// TIA Portal V16 export
// export: Created 2020-08-26T14:42:00.343357Z, ExportSetting WithDefaults, DisplayName Totally Integrated Automation Portal, DisplayVersion V16 Update 2, DisplayName TIA Portal Version Control Interface, DisplayVersion V16 Update 2, DisplayName TIA Portal Openness, DisplayVersion V16 Update 2, DisplayName TIA Portal Teamcenter Gateway, DisplayVersion V16, DisplayName SINAMICS Startdrive Advanced, DisplayVersion V16 Update 1, DisplayName SINAMICS Startdrive G130, G150, S120, S150, SINAMICS MV, S210, DisplayVersion V16 Update 1, DisplayName SINAMICS Startdrive G110M, G120, G120C, G120D, G120P, DisplayVersion V16 Update 1, DisplayName STEP 7 Professional, DisplayVersion V16 Update 2, DisplayName SIMATIC Energy Suite, DisplayVersion V16, DisplayName STEP 7 Safety, DisplayVersion V16, DisplayName WinCC Professional, DisplayVersion V16 Update 2
FUNCTION_BLOCK "SimpleMotor"   // FB2, LAD
{ S7_Optimized_Access := 'TRUE' }
VERSION : 0.1
// stored: AutoNumber true, IsIECCheckEnabled false, IsRetainMemResEnabled false, MemoryReserve 100, SetENOAutomatically false, UDAEnableTagReadback false
   VAR_INPUT
      Start : Bool;
      Stop : Bool;
      Overload : Bool;
      Fault : Bool;
      Reset : Bool;
   END_VAR
   VAR_OUTPUT
      StartCommand : Bool;
   END_VAR
   VAR
      M1Holding : Bool;
      Faulted : Bool;
   END_VAR
BEGIN

REGION Network 1: Start/Stop Network
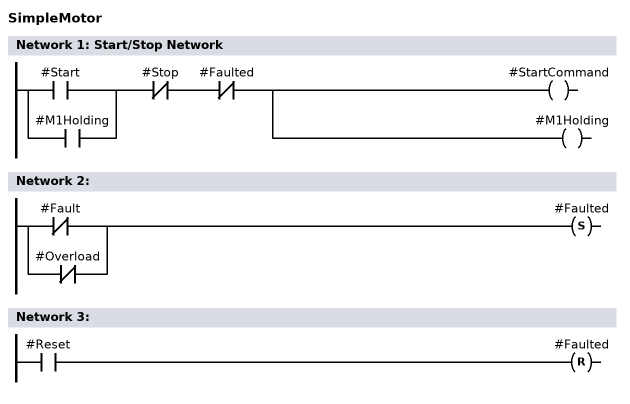
   RUNG wire#powerrail
      Contact( #Start )
      wire#w1
      I_Contact( #Stop )
      I_Contact( #Faulted )
      wire#w2
      Coil( #StartCommand )
   END_RUNG
   RUNG wire#powerrail
      Contact( #M1Holding )
   END_RUNG wire#w1
   RUNG wire#w2
      Coil( #M1Holding )
   END_RUNG
   // the same network as SCL:
   #StartCommand := (#Start OR #M1Holding) AND NOT #Stop AND NOT #Faulted;
   #M1Holding := #StartCommand;
END_REGION

REGION Network 2
   RUNG wire#powerrail
      I_Contact( #Fault )
      wire#w1
      S_Coil( #Faulted )
   END_RUNG
   RUNG wire#powerrail
      I_Contact( #Overload )
   END_RUNG wire#w1
   // the same network as SCL:
   IF NOT #Fault OR NOT #Overload THEN #Faulted := TRUE; END_IF;
END_REGION

REGION Network 3
   RUNG wire#powerrail
      Contact( #Reset )
      R_Coil( #Faulted )
   END_RUNG
   // the same network as SCL:
   IF #Reset THEN #Faulted := FALSE; END_IF;
END_REGION
END_FUNCTION_BLOCK
